// Mitsubishi GX Works2 project: plc1008_factory_count   PLC: Q02/Q02H

PROGRAM MAIN
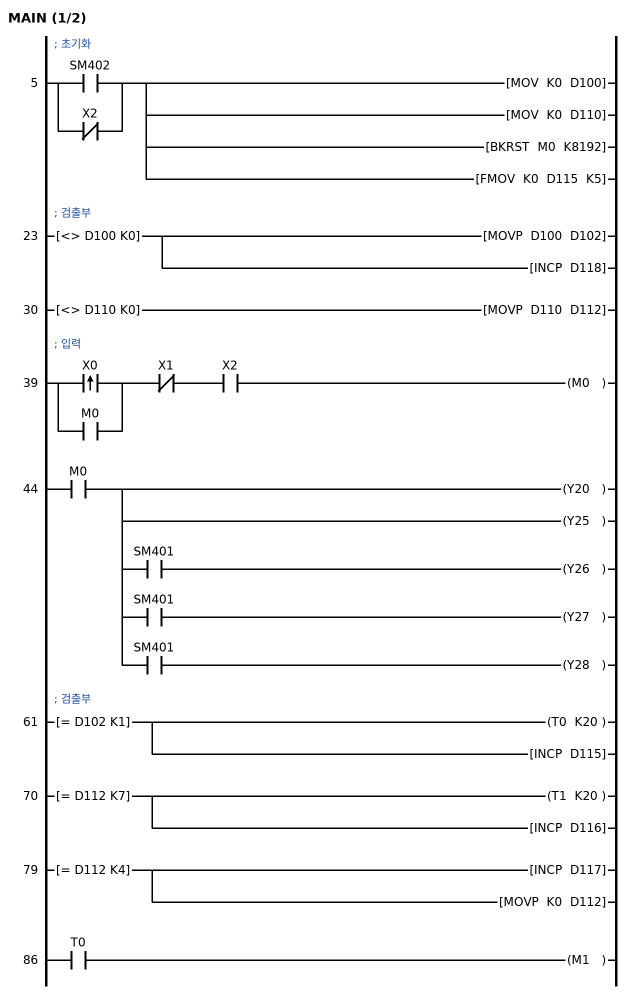
; 초기화
5     LD      SM402
      ORI     X2
      MOV     K0 D100
      MOV     K0 D110
      BKRST   M0 K8192
      FMOV    K0 D115 K5
; 검출부
23    LD<>    D100 K0
      MOVP    D100 D102
      INCP    D118
30    LD<>    D110 K0
      MOVP    D110 D112
; 입력
39    LDP     X0
      OR      M0
      ANI     X1
      AND     X2
      OUT     M0
44    LD      M0
      OUT     Y20
      OUT     Y25
      MPS
      AND     SM401
      OUT     Y26
      MRD
      AND     SM401
      OUT     Y27
      MPP
      AND     SM401
      OUT     Y28
; 검출부
61    LD=     D102 K1
      OUT     T0 K20
      INCP    D115
70    LD=     D112 K7
      OUT     T1 K20
      INCP    D116
79    LD=     D112 K4
      INCP    D117
      MOVP    K0 D112
86    LD      T0
      OUT     M1
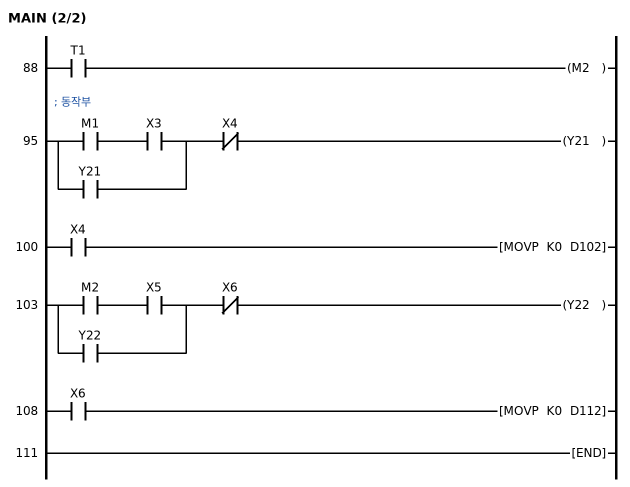
88    LD      T1
      OUT     M2
; 동작부
95    LD      M1
      AND     X3
      OR      Y21
      ANI     X4
      OUT     Y21
100   LD      X4
      MOVP    K0 D102
103   LD      M2
      AND     X5
      OR      Y22
      ANI     X6
      OUT     Y22
108   LD      X6
      MOVP    K0 D112
111   END
END_PROGRAM
